(* CODESYS project EX2.project

Project tree, tasks and I/O mapping:
  Device : CODESYS Control Win V3, 3S - Smart Software Solutions GmbH, order no. 305021, version 3.5.11.30
    application Application
      libraries: Standard, * (System)
      task MainTask (cyclic, interval t#20ms, priority 1) calls PLC_PRG
      program PLC_PRG [LD]
*)

// Device/Application/PLC_PRG
PROGRAM PLC_PRG
VAR
	A : BOOL;               // ENTRADA A
	B : BOOL;               // ENTRADA B
	C : BOOL;               // ENTRADA C
	SAIDA : BOOL;           // SAIDA FINAL
	S1 : BOOL;              // SAIDA         
    S2 : BOOL;              // SAIDA
	S3 : BOOL;              // SAIDA
	S4: BOOL;               // SAIDA
END_VAR

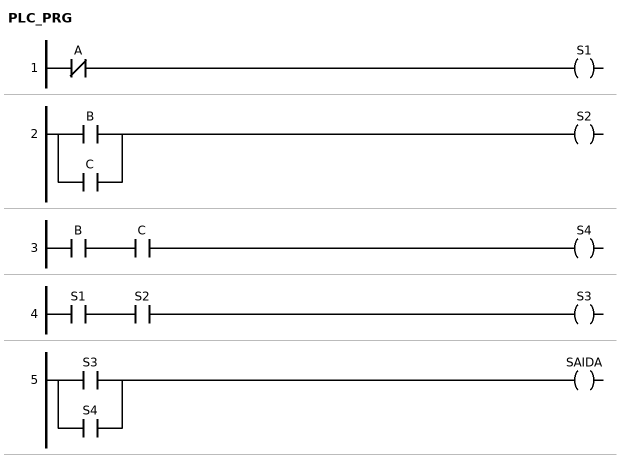
// NETWORK 1
S1 := NOT A;

// NETWORK 2
S2 := B OR C;

// NETWORK 3
S4 := B AND C;

// NETWORK 4
S3 := S1 AND S2;

// NETWORK 5
SAIDA := S3 OR S4;

END_PROGRAM
